Universal Robots PolyScope program: b_watering3.urp

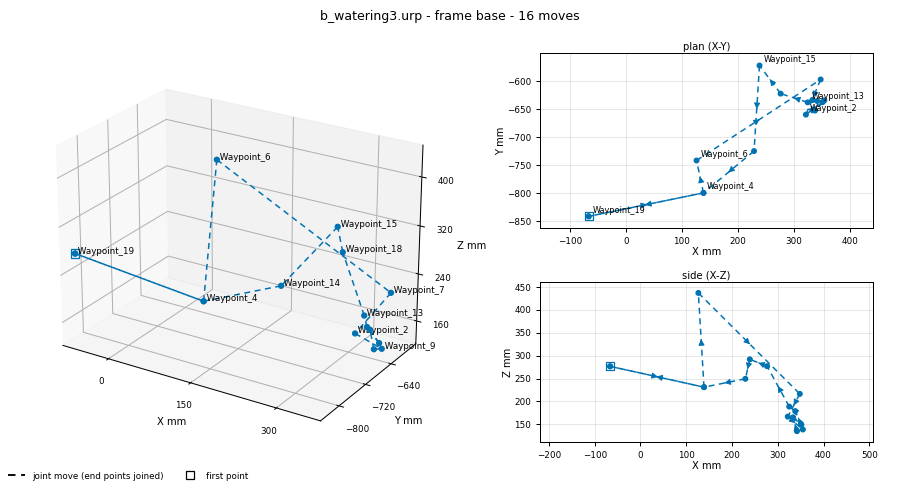
[picture p0: tool path of b_watering3.urp in frame base, 16 of 16 moves have a stored position in this frame; points joined in program order, loops and branches not executed]
Program b_watering3 (installation=default directory=/programs/Burkat_U_Plant createdIn=5.12.6.1102099 lastSavedIn=5.12.6.1102099 robotSerialNumber=20215500597)
Calibrated DH parameters: a=[0.000193, -0.066673, -0.391568, -0.000012, 0.00005, 0]; d=[0.162643, -472.05677, 465.132521, 7.058239, 0.099746, 0.099582]; alpha=[1.571116, 0.00089, 0.003862, 1.569269, -1.569248, 0]; deltaTheta=[0, -1.413394, 7.628392, 0.068187, 0, -0.000001]
Robot Program (runOnlyOnce=true)
  MoveJ speed 30 deg/s, acceleration 50 deg/s^2 (useActiveTCP=true) feature=Base
    Waypoint Waypoint_19: TCP in base x=-66.326 y=-841.615 z=276.687 mm, rx=1.6517 ry=-0.0259 rz=-0.093 rad; joints [71.48, -64.638, 86.648, -17.383, 75.945, -3.629] deg; TCP offset x=0 y=0 z=191.5 mm, rx=0 ry=0 rz=0 rad
    Waypoint Waypoint_4: TCP in base x=138.856 y=-799.749 z=231.2 mm, rx=1.6041 ry=0.0092 rz=-0.0841 rad; joints [92.155, -64.421, 95.991, -29.774, 94.997, -3.194] deg
    Waypoint Waypoint_6: motionParameters(jointSpeed=0.087266 jointAcceleration=0.174533 cartesianSpeed=0.25 cartesianAcceleration=1.2); TCP in base x=126.458 y=-741.84 z=437.108 mm, rx=0.3937 ry=-0.6248 rz=1.6727 rad; joints [91.678, -61.026, 104.293, -96.435, 95.97, 99.942] deg
    Waypoint Waypoint_7: TCP in base x=348.223 y=-597.083 z=216.498 mm, rx=1.4884 ry=0.4988 rz=1.9396 rad; joints [83.574, -47.339, 110.81, -158.413, 16.917, 143.298] deg
  MoveJ speed 40 deg/s, acceleration 60 deg/s^2 (useActiveTCP=true) feature=Base
    Waypoint Waypoint_2: TCP in base x=321.842 y=-659.887 z=166.77 mm, rx=1.5151 ry=0.4071 rz=1.8503 rad; joints [81.634, -43.136, 105.056, -141.767, 15.795, 128.28] deg
  MoveJ speed 20 deg/s, acceleration 50 deg/s^2 (useActiveTCP=true) feature=Base
    Waypoint Waypoint_9: TCP in base x=354.857 y=-634.411 z=138.648 mm, rx=2.2336 ry=0.4447 rz=1.5549 rad; joints [84.864, -56.251, 106.127, -148.152, -18.394, 158.471] deg
  MoveJ speed 10 deg/s, acceleration 20 deg/s^2 (useActiveTCP=true) feature=Base
    Waypoint Waypoint_12: motionParameters(jointSpeed=0.087266 jointAcceleration=0.523599 cartesianSpeed=0.25 cartesianAcceleration=1.2); TCP in base x=341.931 y=-635.554 z=134.955 mm, rx=2.6947 ry=0.5704 rz=0.9561 rad; joints [91.949, -64.579, 95.7, -128.794, -50.107, 160.97] deg
    Waypoint Waypoint_16: TCP in base x=333.35 y=-633.861 z=165.247 mm, rx=2.6896 ry=0.7366 rz=0.4785 rad; joints [98.254, -69.793, 94.358, -130.753, -68.736, 160.832] deg
    Waypoint Waypoint_8: TCP in base x=351.661 y=-637.402 z=148.781 mm, rx=2.5401 ry=0.6556 rz=0.9135 rad; joints [92.307, -66.334, 100.203, -139.487, -48.704, 159.437] deg
    Waypoint Waypoint_17: TCP in base x=338.163 y=-652.62 z=178.842 mm, rx=2.1111 ry=0.6624 rz=1.4167 rad; joints [83.575, -59.768, 102.66, -139.423, -19.049, 143.526] deg
  MoveJ speed 20 deg/s, acceleration 40 deg/s^2 (useActiveTCP=true) feature=Base
    Waypoint Waypoint_13: TCP in base x=325.017 y=-637.937 z=188.746 mm, rx=1.8525 ry=0.3429 rz=1.895 rad; joints [80.611, -47.882, 106.79, -166.203, 3.697, 168.201] deg
    Waypoint Waypoint_18: TCP in base x=276.693 y=-622.322 z=276.989 mm, rx=1.4985 ry=0.3347 rz=2.1364 rad; joints [77.642, -47.916, 106.841, -166.244, 22.416, 168.176] deg
  MoveJ speed 30 deg/s, acceleration 60 deg/s^2 (useActiveTCP=true) feature=Base
    Waypoint Waypoint_15: TCP in base x=238.95 y=-572.137 z=292.042 mm, rx=1.1037 ry=0.9926 rz=1.0267 rad; joints [70.17, -58.462, 118.936, -187.558, 12.187, 121.487] deg
    Waypoint Waypoint_14: TCP in base x=229.199 y=-724.969 z=249.427 mm, rx=1.4494 ry=0.0699 rz=1.0404 rad; joints [80.427, -66.589, 109.198, -59.695, 43.195, 45.792] deg
    Waypoint Waypoint_4: TCP in base x=138.856 y=-799.749 z=231.2 mm, rx=1.6041 ry=0.0092 rz=-0.0841 rad; joints [92.155, -64.421, 95.991, -29.774, 94.997, -3.194] deg
    Waypoint Waypoint_19: TCP in base x=-66.326 y=-841.615 z=276.687 mm, rx=1.6517 ry=-0.0259 rz=-0.093 rad; joints [71.48, -64.638, 86.648, -17.383, 75.945, -3.629] deg
